// TIA Portal V18 export
FUNCTION_BLOCK "not_used_blocks"   // FB48, FBD
{ S7_Optimized_Access := 'TRUE' }
VERSION : 0.1
// stored: AutoNumber true, IsIECCheckEnabled false, IsRetainMemResEnabled false, MemoryReserve 100, SetENOAutomatically false, UDAEnableTagReadback false
   VAR
      isMultiturn : Bool;
      MultiTurnGoesFwdOnly : Bool;
      SET_SPD_ABS : Real;
      POS : Real;
      TARGET : Real;
      par_lim_fwd : Real;
      par_lim_rev : Real;
      par_spd_absmax : Real;
      par_dist_absMax : Real;
      par_spd_crawl : Real;
      par_dist_crawl : Real;
      par_dist_stop : Real;
      speed_limited_by_target : Real;
      ER : Bool;
      ER_w : WString;
      mot_universal_arrived_missed_Instance { S7_SetPoint := 'True'} : "mot_universal_arrived_missed";
      was_set : Bool;
   END_VAR
   VAR_TEMP
      rtyui1 : Bool;
   END_VAR
BEGIN

REGION Network 2
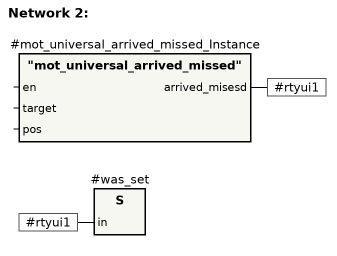
   #mot_universal_arrived_missed_Instance(arrived_misesd => #rtyui1);   // "mot_universal_arrived_missed"
   IF #rtyui1 THEN #was_set := TRUE; END_IF;
END_REGION
END_FUNCTION_BLOCK
